(* Logix 5000 project; controller cal1615 1756-L62 rev 20.19; software revision 20.05; part 60 of 82 *)
(* tags used below, declared in another part *)
   FAULT : BOOL;   // Fault AFI
   HMI : BOOL;   // AFI HMI
   p01r09_pb_global_reset : BOOL;   // System Modes PB: Global Fault Reset
   p25_di_jog : BOOL;   // Tension Stand 2 Digital Input SS: Jog
   p25_di_jog_fwd : BOOL;   // Tension Stand 2 Digital Input PB: Jog Forward
   p25_di_jog_rev : BOOL;   // Tension Stand 2 Digital Input PB: Jog Reverse
   p25_di_run : BOOL;   // Tension Stand 2 Digital Input SS: Run
   p25_dint_to_hmi : DINT[16];   // Tension Stand 2 Dint to HMI
   p25r01 : routine;
   p25r07 : routine;
   p25r07_timer_fault : TIMER[4];   // Tension Stand 2 Alarms Fault Dwell Time
   p25r07_timer_warning : TIMER[4];   // Tension Stand 2 Alarms Warning Dwell Timer
   p25r08 : routine;
   p25r08_timer_fault : TIMER[4];   // Tension Stand 2 Warnings Fault Dwell Timer
   p25r08_timer_warning : TIMER[4];   // Tension Stand 2 Warnings Warning Dwell Timer
   p25r09 : routine;   // Upper Poly Letoff Modes
   p25r09_mode_jog : BOOL;   // Tension Stand 2 Modes Jog Mode
   p25r09_mode_run : BOOL;   // Tension Stand 2 Modes Run Mode
   p25r09_mode_thread : BOOL;   // Tension Stand 2 Modes Thread Mode
   p25r09_pb_jog_fwd : BOOL;   // Tension Stand 2 Modes PB: Jog Forward
   p25r09_pb_jog_rev : BOOL;   // Tension Stand 2 Modes PB: Jog Reverse
   p25r09_timer_fault : TIMER[4];   // Tension Stand 2 Modes Fault Dwell Timer
   p25r09_timer_warning : TIMER[4];   // Tension Stand 2 Modes Warning Dwell Timer
   p25r11 : routine;   // Tension Stand 2 VFD
(* P25_Tension_Stand_2, continued *)

ROUTINE R07_Alarms   (* ladder *)
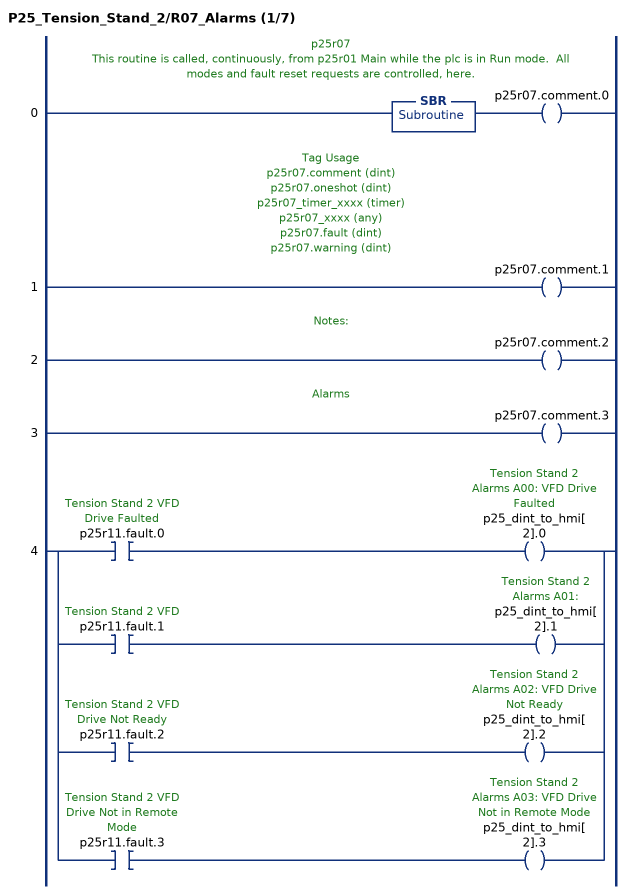
   // p25r07
   // This routine is called, continuously, from p25r01 Main while the plc is in Run mode.  All modes and fault reset requests are controlled, here.
   0: SBR()OTE(p25r07.comment.0);
   // Tag Usage
   // p25r07.comment (dint)
   // p25r07.oneshot (dint)
   // p25r07_timer_xxxx (timer)
   // p25r07_xxxx (any)
   // p25r07.fault (dint)
   // p25r07.warning (dint)
   1: OTE(p25r07.comment.1);
   // Notes:
   2: OTE(p25r07.comment.2);
   // Alarms
   3: OTE(p25r07.comment.3);
   4: [XIC(p25r11.fault.0) OTE(p25_dint_to_hmi[2].0) ,XIC(p25r11.fault.1) OTE(p25_dint_to_hmi[2].1) ,XIC(p25r11.fault.2) OTE(p25_dint_to_hmi[2].2) ,XIC(p25r11.fault.3) OTE(p25_dint_to_hmi[2].3) ];
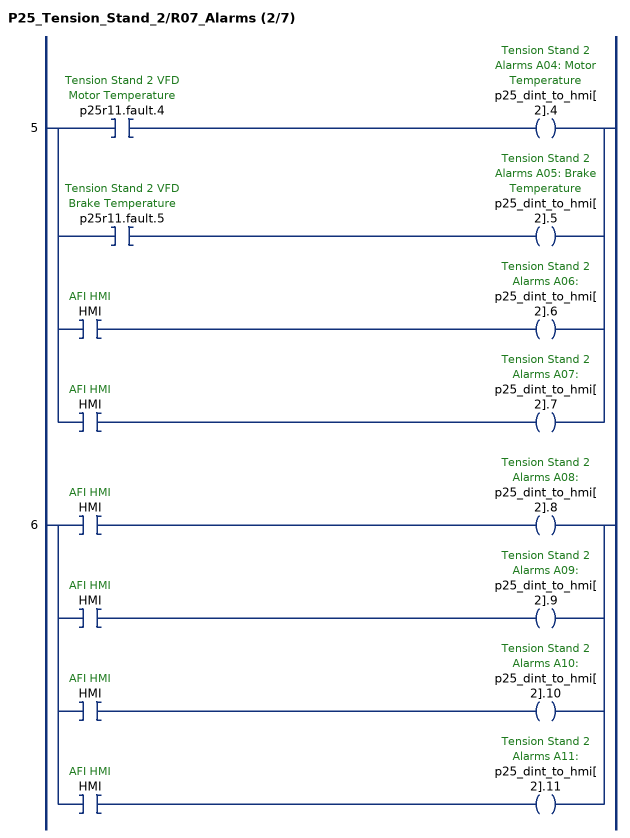
   5: [XIC(p25r11.fault.4) OTE(p25_dint_to_hmi[2].4) ,XIC(p25r11.fault.5) OTE(p25_dint_to_hmi[2].5) ,XIC(HMI) OTE(p25_dint_to_hmi[2].6) ,XIC(HMI) OTE(p25_dint_to_hmi[2].7) ];
   6: [XIC(HMI) OTE(p25_dint_to_hmi[2].8) ,XIC(HMI) OTE(p25_dint_to_hmi[2].9) ,XIC(HMI) OTE(p25_dint_to_hmi[2].10) ,XIC(HMI) OTE(p25_dint_to_hmi[2].11) ];
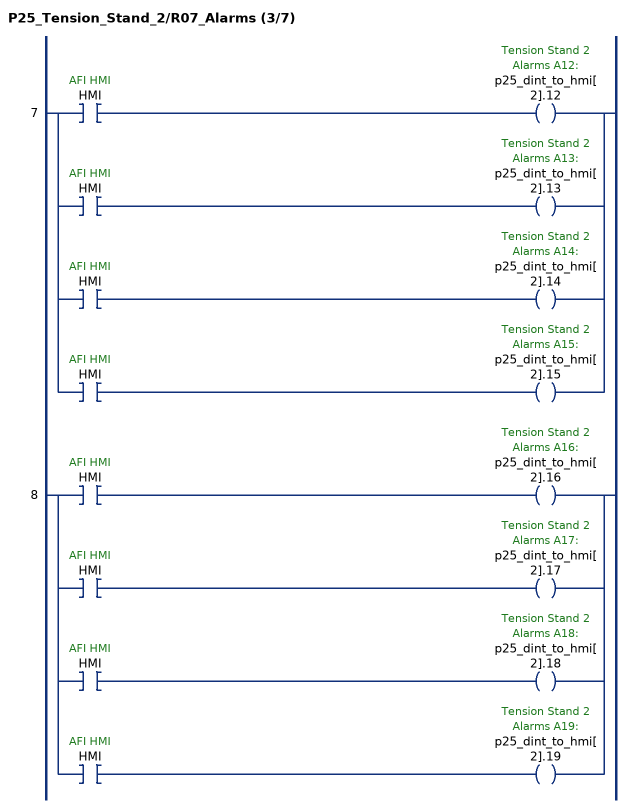
   7: [XIC(HMI) OTE(p25_dint_to_hmi[2].12) ,XIC(HMI) OTE(p25_dint_to_hmi[2].13) ,XIC(HMI) OTE(p25_dint_to_hmi[2].14) ,XIC(HMI) OTE(p25_dint_to_hmi[2].15) ];
   8: [XIC(HMI) OTE(p25_dint_to_hmi[2].16) ,XIC(HMI) OTE(p25_dint_to_hmi[2].17) ,XIC(HMI) OTE(p25_dint_to_hmi[2].18) ,XIC(HMI) OTE(p25_dint_to_hmi[2].19) ];
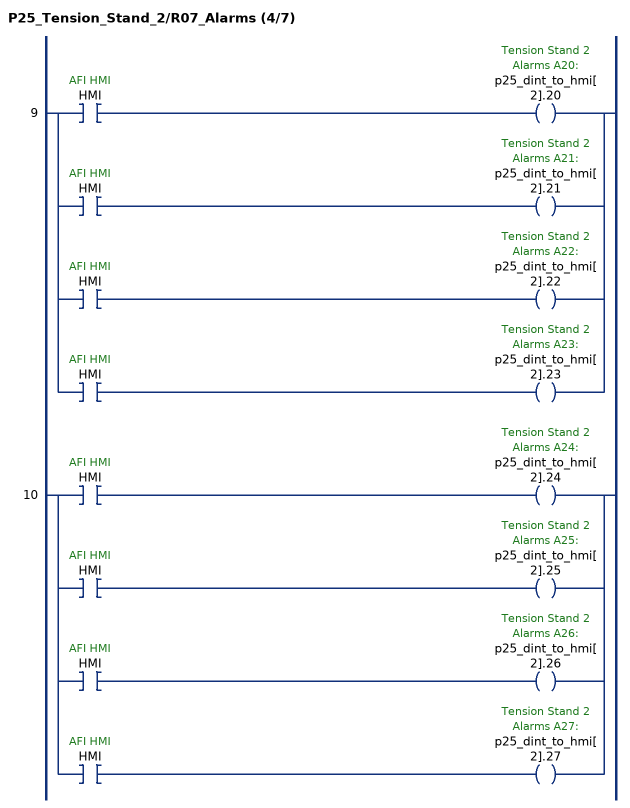
   9: [XIC(HMI) OTE(p25_dint_to_hmi[2].20) ,XIC(HMI) OTE(p25_dint_to_hmi[2].21) ,XIC(HMI) OTE(p25_dint_to_hmi[2].22) ,XIC(HMI) OTE(p25_dint_to_hmi[2].23) ];
   10: [XIC(HMI) OTE(p25_dint_to_hmi[2].24) ,XIC(HMI) OTE(p25_dint_to_hmi[2].25) ,XIC(HMI) OTE(p25_dint_to_hmi[2].26) ,XIC(HMI) OTE(p25_dint_to_hmi[2].27) ];
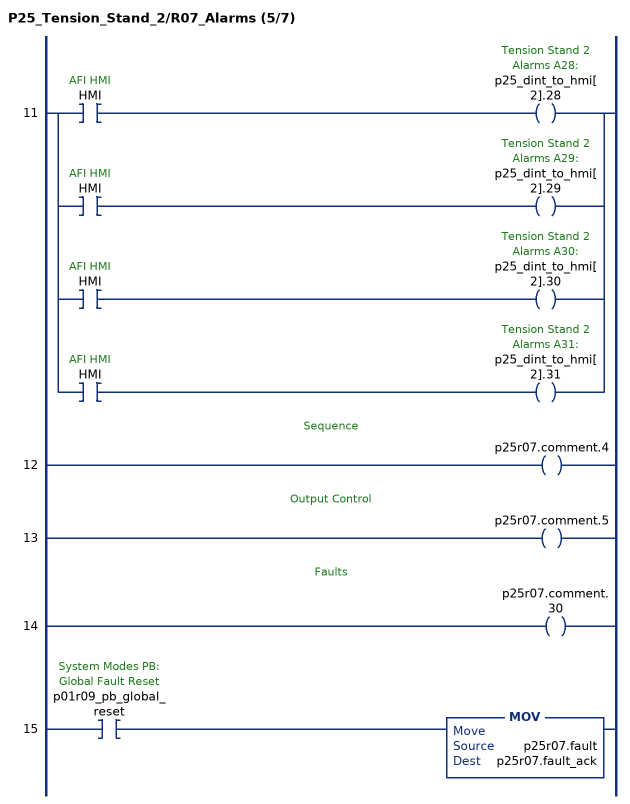
   11: [XIC(HMI) OTE(p25_dint_to_hmi[2].28) ,XIC(HMI) OTE(p25_dint_to_hmi[2].29) ,XIC(HMI) OTE(p25_dint_to_hmi[2].30) ,XIC(HMI) OTE(p25_dint_to_hmi[2].31) ];
   // Sequence
   12: OTE(p25r07.comment.4);
   // Output Control
   13: OTE(p25r07.comment.5);
   // Faults
   14: OTE(p25r07.comment.30);
   15: XIC(p01r09_pb_global_reset)MOV(p25r07.fault,p25r07.fault_ack);
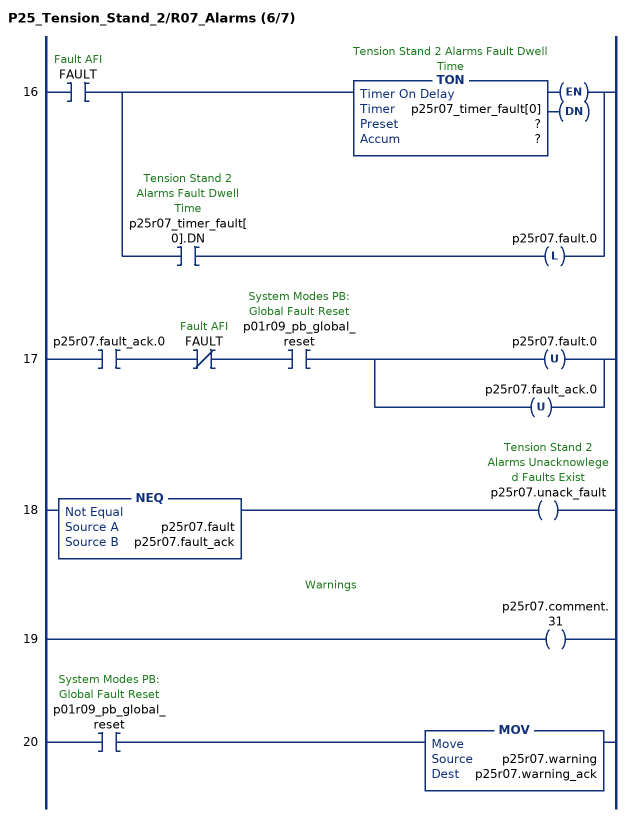
   16: XIC(FAULT)[TON(p25r07_timer_fault[0],?,?) ,XIC(p25r07_timer_fault[0].DN) OTL(p25r07.fault.0) ];
   17: XIC(p25r07.fault_ack.0)XIO(FAULT)XIC(p01r09_pb_global_reset)[OTU(p25r07.fault.0) ,OTU(p25r07.fault_ack.0) ];
   18: NEQ(p25r07.fault,p25r07.fault_ack)OTE(p25r07.unack_fault);
   // Warnings
   19: OTE(p25r07.comment.31);
   20: XIC(p01r09_pb_global_reset)MOV(p25r07.warning,p25r07.warning_ack);
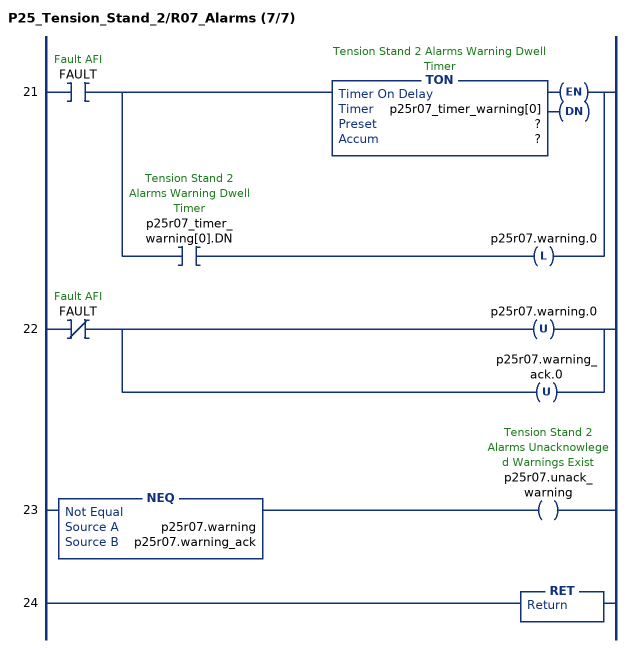
   21: XIC(FAULT)[TON(p25r07_timer_warning[0],?,?) ,XIC(p25r07_timer_warning[0].DN) OTL(p25r07.warning.0) ];
   22: XIO(FAULT)[OTU(p25r07.warning.0) ,OTU(p25r07.warning_ack.0) ];
   23: NEQ(p25r07.warning,p25r07.warning_ack)OTE(p25r07.unack_warning);
   24: RET();
END_ROUTINE

ROUTINE R08_Warnings   (* ladder *)
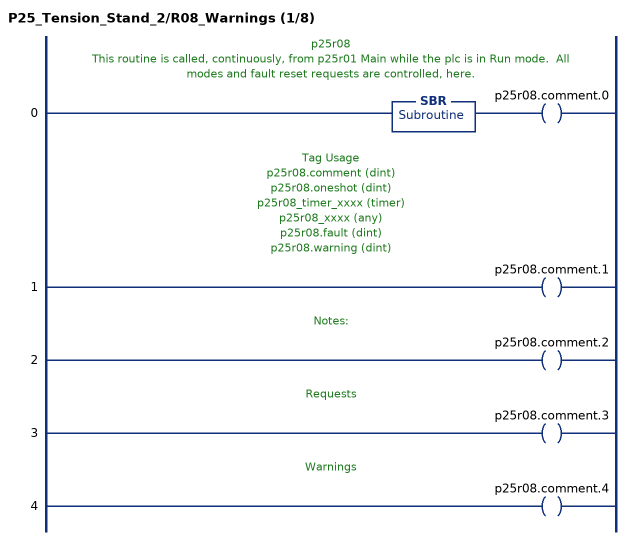
   // p25r08
   // This routine is called, continuously, from p25r01 Main while the plc is in Run mode.  All modes and fault reset requests are controlled, here.
   0: SBR()OTE(p25r08.comment.0);
   // Tag Usage
   // p25r08.comment (dint)
   // p25r08.oneshot (dint)
   // p25r08_timer_xxxx (timer)
   // p25r08_xxxx (any)
   // p25r08.fault (dint)
   // p25r08.warning (dint)
   1: OTE(p25r08.comment.1);
   // Notes:
   2: OTE(p25r08.comment.2);
   // Requests
   3: OTE(p25r08.comment.3);
   // Warnings
   4: OTE(p25r08.comment.4);
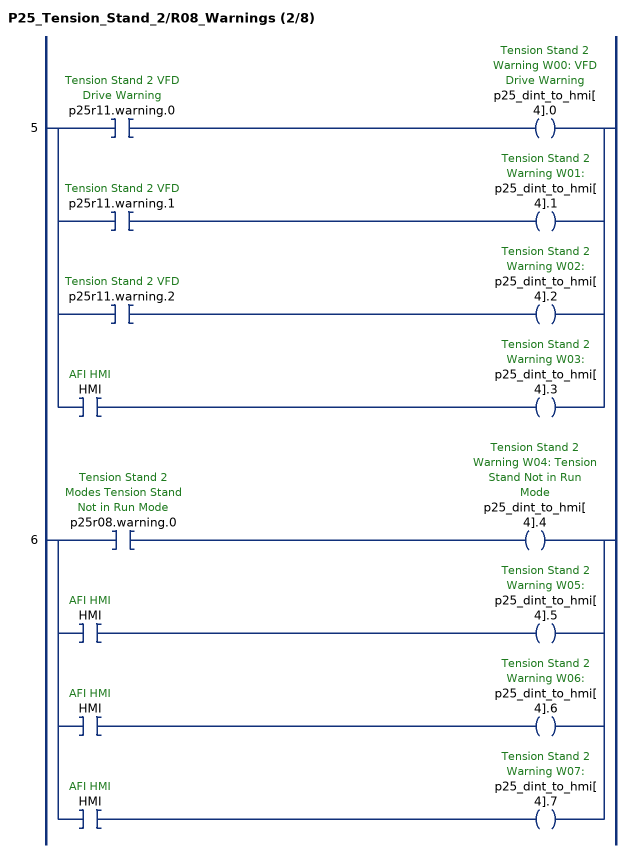
   5: [XIC(p25r11.warning.0) OTE(p25_dint_to_hmi[4].0) ,XIC(p25r11.warning.1) OTE(p25_dint_to_hmi[4].1) ,XIC(p25r11.warning.2) OTE(p25_dint_to_hmi[4].2) ,XIC(HMI) OTE(p25_dint_to_hmi[4].3) ];
   6: [XIC(p25r08.warning.0) OTE(p25_dint_to_hmi[4].4) ,XIC(HMI) OTE(p25_dint_to_hmi[4].5) ,XIC(HMI) OTE(p25_dint_to_hmi[4].6) ,XIC(HMI) OTE(p25_dint_to_hmi[4].7) ];
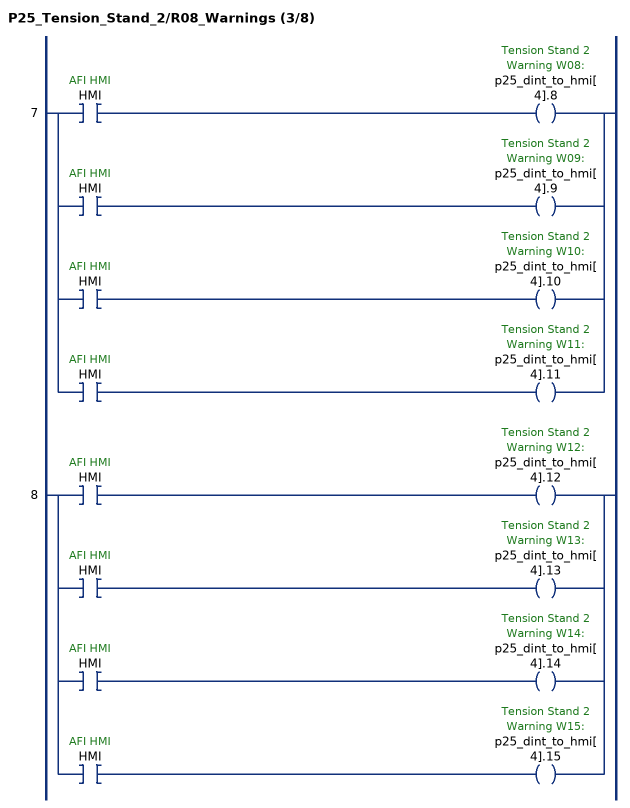
   7: [XIC(HMI) OTE(p25_dint_to_hmi[4].8) ,XIC(HMI) OTE(p25_dint_to_hmi[4].9) ,XIC(HMI) OTE(p25_dint_to_hmi[4].10) ,XIC(HMI) OTE(p25_dint_to_hmi[4].11) ];
   8: [XIC(HMI) OTE(p25_dint_to_hmi[4].12) ,XIC(HMI) OTE(p25_dint_to_hmi[4].13) ,XIC(HMI) OTE(p25_dint_to_hmi[4].14) ,XIC(HMI) OTE(p25_dint_to_hmi[4].15) ];
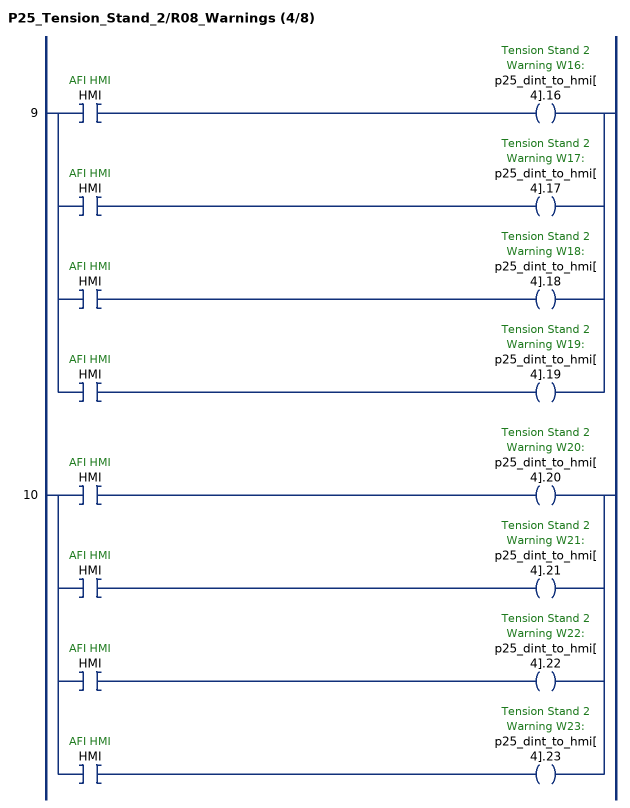
   9: [XIC(HMI) OTE(p25_dint_to_hmi[4].16) ,XIC(HMI) OTE(p25_dint_to_hmi[4].17) ,XIC(HMI) OTE(p25_dint_to_hmi[4].18) ,XIC(HMI) OTE(p25_dint_to_hmi[4].19) ];
   10: [XIC(HMI) OTE(p25_dint_to_hmi[4].20) ,XIC(HMI) OTE(p25_dint_to_hmi[4].21) ,XIC(HMI) OTE(p25_dint_to_hmi[4].22) ,XIC(HMI) OTE(p25_dint_to_hmi[4].23) ];
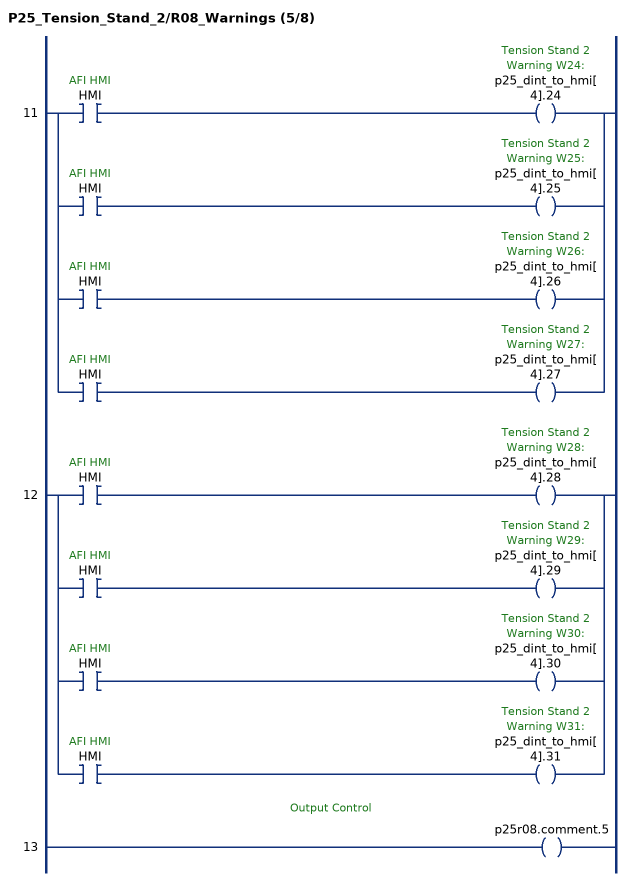
   11: [XIC(HMI) OTE(p25_dint_to_hmi[4].24) ,XIC(HMI) OTE(p25_dint_to_hmi[4].25) ,XIC(HMI) OTE(p25_dint_to_hmi[4].26) ,XIC(HMI) OTE(p25_dint_to_hmi[4].27) ];
   12: [XIC(HMI) OTE(p25_dint_to_hmi[4].28) ,XIC(HMI) OTE(p25_dint_to_hmi[4].29) ,XIC(HMI) OTE(p25_dint_to_hmi[4].30) ,XIC(HMI) OTE(p25_dint_to_hmi[4].31) ];
   // Output Control
   13: OTE(p25r08.comment.5);
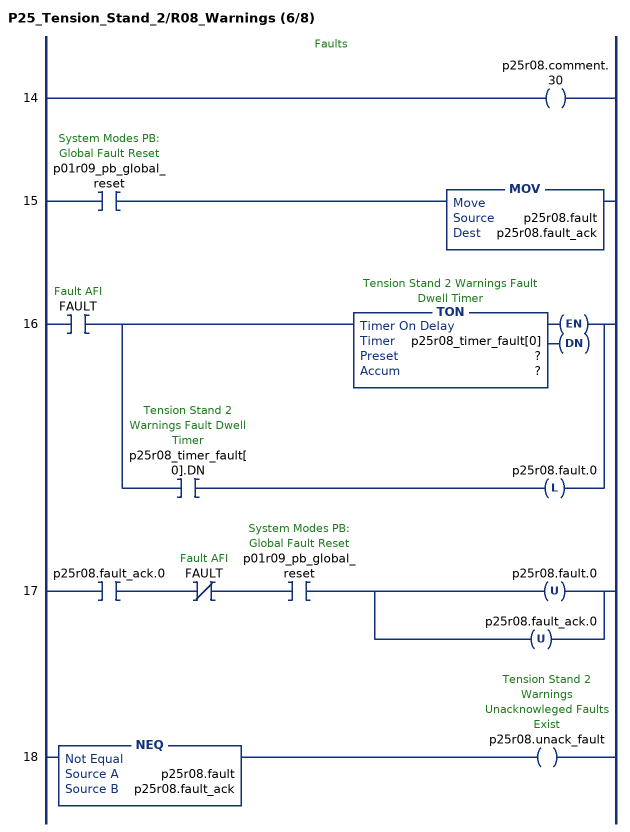
   // Faults
   14: OTE(p25r08.comment.30);
   15: XIC(p01r09_pb_global_reset)MOV(p25r08.fault,p25r08.fault_ack);
   16: XIC(FAULT)[TON(p25r08_timer_fault[0],?,?) ,XIC(p25r08_timer_fault[0].DN) OTL(p25r08.fault.0) ];
   17: XIC(p25r08.fault_ack.0)XIO(FAULT)XIC(p01r09_pb_global_reset)[OTU(p25r08.fault.0) ,OTU(p25r08.fault_ack.0) ];
   18: NEQ(p25r08.fault,p25r08.fault_ack)OTE(p25r08.unack_fault);
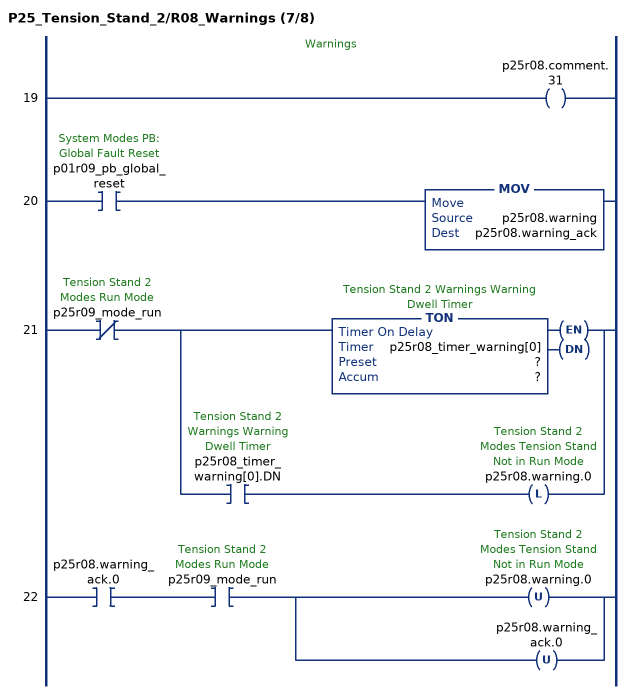
   // Warnings
   19: OTE(p25r08.comment.31);
   20: XIC(p01r09_pb_global_reset)MOV(p25r08.warning,p25r08.warning_ack);
   21: XIO(p25r09_mode_run)[TON(p25r08_timer_warning[0],?,?) ,XIC(p25r08_timer_warning[0].DN) OTL(p25r08.warning.0) ];
   22: XIC(p25r08.warning_ack.0)XIC(p25r09_mode_run)[OTU(p25r08.warning.0) ,OTU(p25r08.warning_ack.0) ];
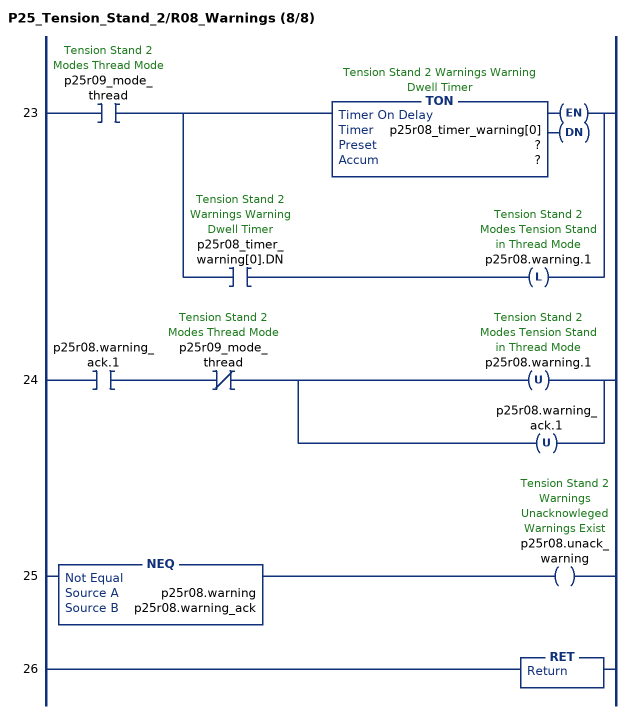
   23: XIC(p25r09_mode_thread)[TON(p25r08_timer_warning[0],?,?) ,XIC(p25r08_timer_warning[0].DN) OTL(p25r08.warning.1) ];
   24: XIC(p25r08.warning_ack.1)XIO(p25r09_mode_thread)[OTU(p25r08.warning.1) ,OTU(p25r08.warning_ack.1) ];
   25: NEQ(p25r08.warning,p25r08.warning_ack)OTE(p25r08.unack_warning);
   26: RET();
END_ROUTINE

ROUTINE R09_Modes   (* ladder *)
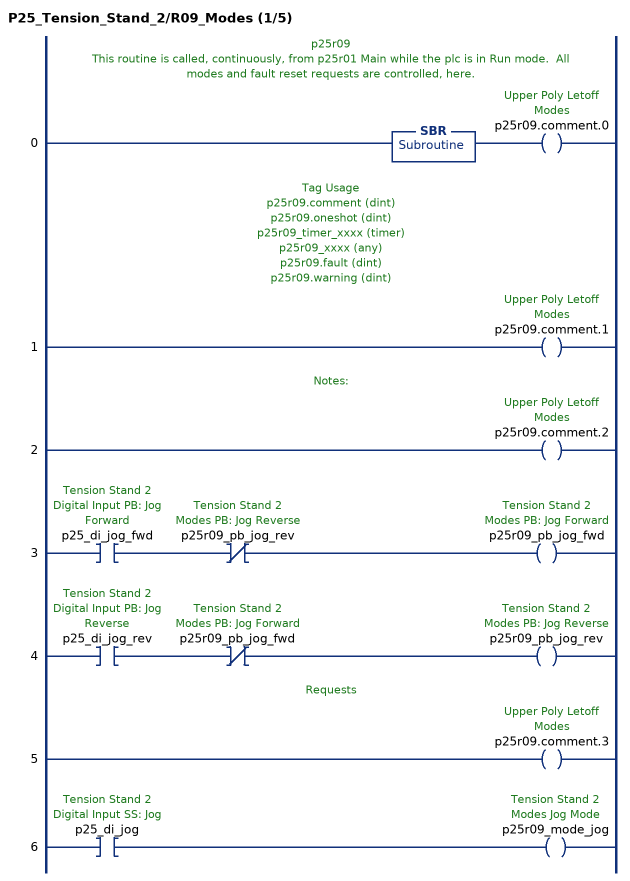
   // p25r09
   // This routine is called, continuously, from p25r01 Main while the plc is in Run mode.  All modes and fault reset requests are controlled, here.
   0: SBR()OTE(p25r09.comment.0);
   // Tag Usage
   // p25r09.comment (dint)
   // p25r09.oneshot (dint)
   // p25r09_timer_xxxx (timer)
   // p25r09_xxxx (any)
   // p25r09.fault (dint)
   // p25r09.warning (dint)
   1: OTE(p25r09.comment.1);
   // Notes:
   2: OTE(p25r09.comment.2);
   3: XIC(p25_di_jog_fwd)XIO(p25r09_pb_jog_rev)OTE(p25r09_pb_jog_fwd);
   4: XIC(p25_di_jog_rev)XIO(p25r09_pb_jog_fwd)OTE(p25r09_pb_jog_rev);
   // Requests
   5: OTE(p25r09.comment.3);
   6: XIC(p25_di_jog)OTE(p25r09_mode_jog);
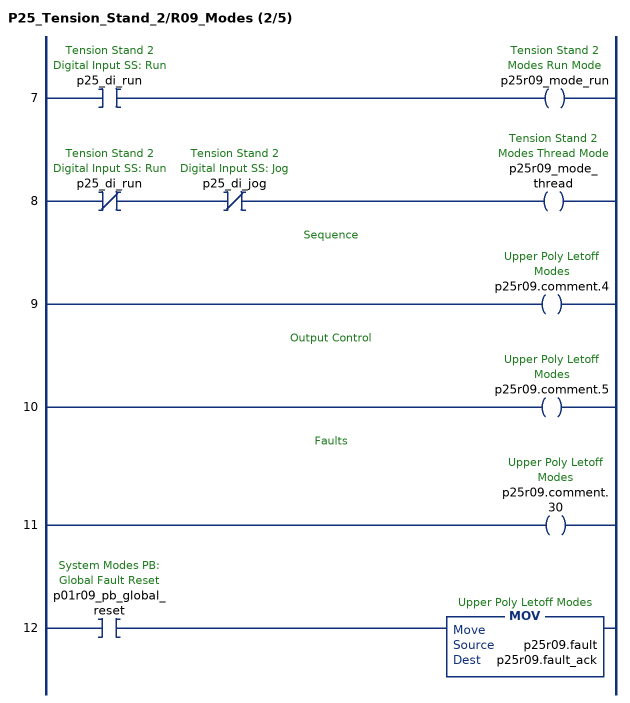
   7: XIC(p25_di_run)OTE(p25r09_mode_run);
   8: XIO(p25_di_run)XIO(p25_di_jog)OTE(p25r09_mode_thread);
   // Sequence
   9: OTE(p25r09.comment.4);
   // Output Control
   10: OTE(p25r09.comment.5);
   // Faults
   11: OTE(p25r09.comment.30);
   12: XIC(p01r09_pb_global_reset)MOV(p25r09.fault,p25r09.fault_ack);
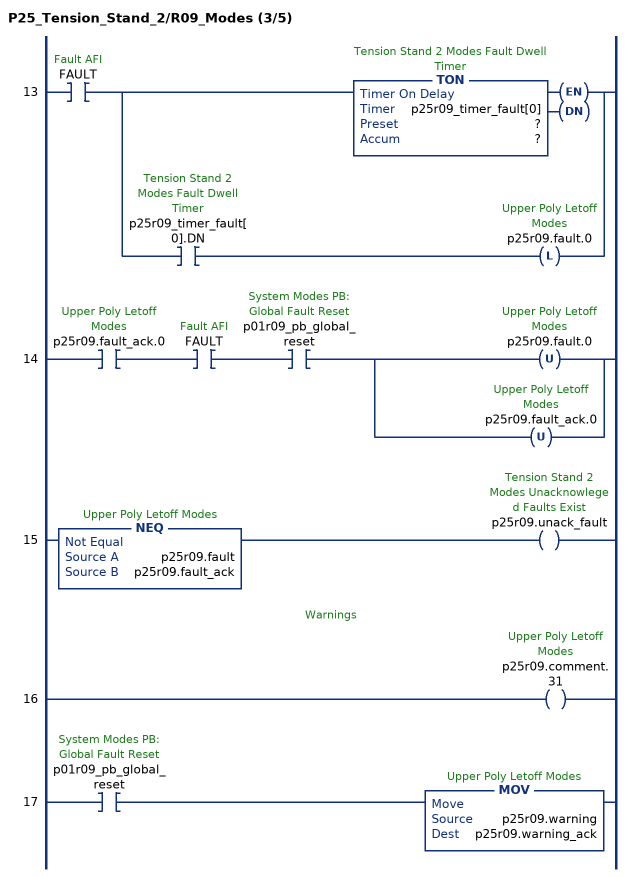
   13: XIC(FAULT)[TON(p25r09_timer_fault[0],?,?) ,XIC(p25r09_timer_fault[0].DN) OTL(p25r09.fault.0) ];
   14: XIC(p25r09.fault_ack.0)XIC(FAULT)XIC(p01r09_pb_global_reset)[OTU(p25r09.fault.0) ,OTU(p25r09.fault_ack.0) ];
   15: NEQ(p25r09.fault,p25r09.fault_ack)OTE(p25r09.unack_fault);
   // Warnings
   16: OTE(p25r09.comment.31);
   17: XIC(p01r09_pb_global_reset)MOV(p25r09.warning,p25r09.warning_ack);
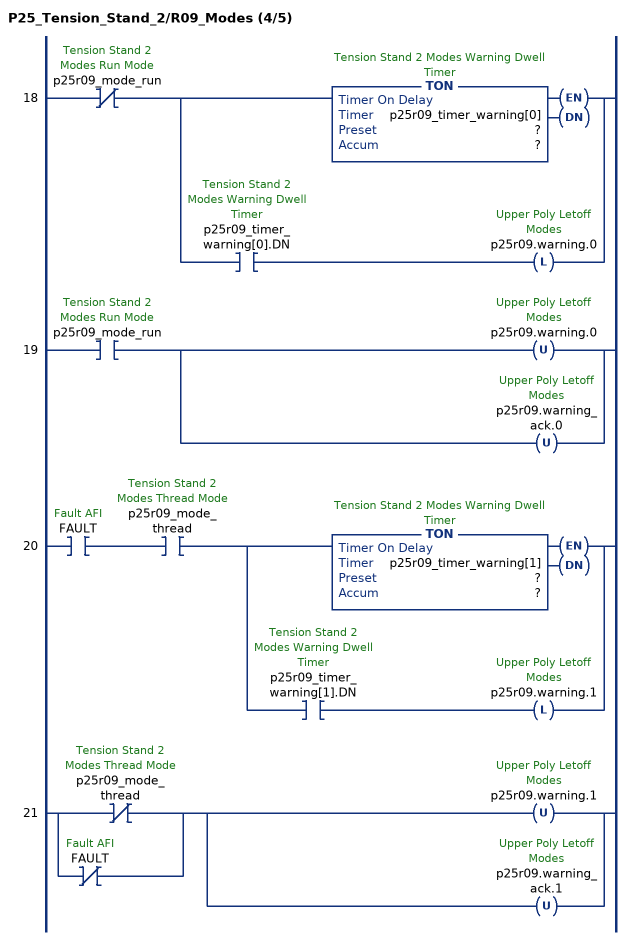
   18: XIO(p25r09_mode_run)[TON(p25r09_timer_warning[0],?,?) ,XIC(p25r09_timer_warning[0].DN) OTL(p25r09.warning.0) ];
   19: XIC(p25r09_mode_run)[OTU(p25r09.warning.0) ,OTU(p25r09.warning_ack.0) ];
   20: XIC(FAULT)XIC(p25r09_mode_thread)[TON(p25r09_timer_warning[1],?,?) ,XIC(p25r09_timer_warning[1].DN) OTL(p25r09.warning.1) ];
   21: [XIO(p25r09_mode_thread) ,XIO(FAULT) ][OTU(p25r09.warning.1) ,OTU(p25r09.warning_ack.1) ];
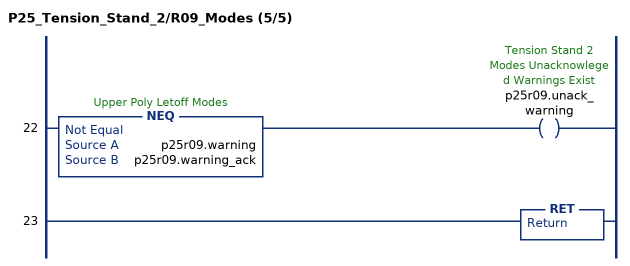
   22: NEQ(p25r09.warning,p25r09.warning_ack)OTE(p25r09.unack_warning);
   23: RET();
END_ROUTINE
